// Frees pointer when this instance of the FB leaves the scope;
{attribute 'no_explicit_call' := 'do not call this POU directly'}
FUNCTION_BLOCK INTERNAL FINAL FB_Free
VAR
	pValue : REFERENCE TO POINTER TO BYTE;
END_VAR

METHOD FB_exit : BOOL
VAR_INPUT
	bInCopyCode : BOOL; // if TRUE, the exit method is called for exiting an instance that is copied afterwards (online change).
END_VAR
IF NOT __ISVALIDREF(THIS^.pValue) THEN RETURN; END_IF
IF THIS^.pValue <> 0 THEN __DELETE(THIS^.pValue); END_IF
END_METHOD

{attribute 'no_explicit_call' := 'do not call this POU directly'}
METHOD FB_init : BOOL
VAR_INPUT
	bInitRetains 	: BOOL; // if TRUE, the retain variables are initialized (warm start / cold start)
	bInCopyCode 	: BOOL;  // if TRUE, the instance afterwards gets moved into the copy code (online change)
	pValue 			: REFERENCE TO POINTER TO BYTE; // Pointer to be freed on exit
END_VAR
THIS^.pValue REF= pValue;
END_METHOD

END_FUNCTION_BLOCK

(* stored: Version 1.1.0.1, ProductVersion 3.1.4024.4
   POU FB_Free: Id {0f81eb6c-8fe8-40d5-bea2-24b57eb73072}, SpecialFunc None
   Method FB_exit: Id {6935ded8-4653-46a1-a1bb-b2ee7b43a0a8}
   Method FB_init: Id {b3c81f82-ab5d-4cdf-8e5d-722eff5ef3e8} *)
